// Mitsubishi GX Works2 project: 230927-006-A1.A2   PLC: Q03UDV

// task Task_01 (event TRUE, interval 0, priority 31): POU_01

PROGRAM POU_01
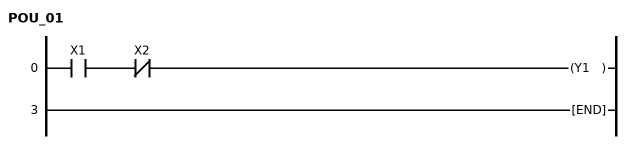
0     LD      X1
      ANI     X2
      OUT     Y1
3     END
END_PROGRAM
